(* PLC project faults, TNI-Software ControlBuild 4.00.18 *)
(* stored: creationDateTime 2005-06-22T10:04:44-01:00 *)

FUNCTION_BLOCK batch.faults
  VAR_INPUT  (* CB.kind=inputVars *)
    fault3 : BOOL := false;
    fault2 : BOOL := false;
    fault1 : BOOL := false;
  END_VAR
  VAR_OUTPUT  (* CB.kind=outputVars *)
    generalFault : BOOL := false;  (* CB.mnemonicPatternPropertyName=generalFault<SY><NU> *)
  END_VAR

(* LD diagram, written out as Structured Text *)
1:
generalFault := fault3 OR fault1 OR fault2;
END_FUNCTION_BLOCK
